// TIA Portal project "Simulacaoportao" (V14)
// Simulação do projeto portao

(* hardware
DEVICE "S7-1200 station_1"  S7-1200 Station
   slot 0: "Rack_0"  S7-1200 Rack  Rack  V1.0
   slot 1: "PLC_1"  CPU 1214C DC/DC/DC  6ES7 214-1AG40-0XB0  V4.2
*)

// ===== PLC "PLC_1"  CPU 1214C DC/DC/DC =====

VAR_GLOBAL   // PLC tag table "Default tag table"
   ""BotaoAbrir"" AT %I0.1 : Bool;
   ""BotaoFechar"" AT %I0.2 : Bool;
   ""SensorPortaAberta"" AT %I0.3 : Bool;
   ""SensorPortaFechada"" AT %I0.4 : Bool;
   ""SensorInfravermelhoSeg"" AT %I0.5 : Bool;
   ""MotorAbrePortao"" AT %Q0.1 : Bool;
   ""MotorFechaPortao"" AT %Q0.2 : Bool;
END_VAR